Staubli VAL3: unSelectItem.pgx

program unSelectItem()
  local string l_sEvent
  local num i
  local num l_nSize
begin
end
